// TwinCAT 3 PLC project PLC_HMI
// ProgramVersion: 3.1.4024.0
// libraries:
//   CmpBitmapPool, * (System)
//   Tc2_Standard, * (Beckhoff Automation GmbH)
//   Tc2_System, * (Beckhoff Automation GmbH)
//   Tc2_Utilities, * (Beckhoff Automation GmbH)
//   Tc3_Module, * (Beckhoff Automation GmbH)
//   VisuDialogs, * (System)
// project tree:
//   / GlobalTextList.TcGTLO, PlcTask.TcTTO, VisualizationManager.TcVMO (not stored), VISU_TASK.TcTTO
//   GVLs/ GVL.TcGVL
//   POUs/ FB_UpdateTimeStamp.TcPOU, MAIN.TcPOU, OP_BTN.TcPOU
//   VISUs/ CONFIRMATION.TcVIS, FOOTER.TcVIS, PAGE_SYSTEM.TcVIS, PAGE_RUN.TcVIS, ImagePool.TcIPO (not stored), PAGE_HOME.TcVIS, PAGE_CONTROL.TcVIS
// real-time tasks:
//   TASK PlcTask: cycle T#10ms, priority 20, ADS port 350
//   TASK VISU_TASK: cycle T#200000us, priority 30, ADS port 351

CONFIGURATION PLC_HMI
    RESOURCE PLC ON TwinCAT3
        TASK PlcTask(INTERVAL := T#10ms, PRIORITY := 20);
        TASK VISU_TASK(INTERVAL := T#200000us, PRIORITY := 30);
        PROGRAM MAIN WITH PlcTask : MAIN;
        PROGRAM VisuElems_Visu_Prg WITH VISU_TASK : VisuElems.Visu_Prg;
    END_RESOURCE
END_CONFIGURATION

// ---- GVLs/GVL.TcGVL
{attribute 'qualified_only'}
VAR_GLOBAL
	TableRecord		: ARRAY [1..5,1..7] OF STRING;
	TODAY			: WORD;
	YESTERDAY		: WORD;
	LASTMONTH		: UINT;
	LASTYEAR		: UINT;
	
	DailyCnt_FG1	: INT;
	DailyCnt_FG2	: INT;
	DailyCnt_FG3	: INT;
	DailyCnt_FG4	: INT;
	MonthCnt		: UINT;
	YearCnt			: UINT;
END_VAR

// ---- POUs/MAIN.TcPOU
PROGRAM MAIN
VAR
	fb_TimeStamp : FB_UpdateTimeStamp ();
END_VAR

// Open PLC HMI view here C:\TwinCAT\3.1\Components\Plc\Tc3PlcHmi
// Open PLC HMI web view with this link   http://127.0.0.1/Tc3PlcHmiWeb/Port_851/Visu/webvisu.htm


fb_TimeStamp();
OP_BTN();

END_PROGRAM

// ---- POUs/FB_UpdateTimeStamp.TcPOU
FUNCTION_BLOCK FB_UpdateTimeStamp
VAR_INPUT
END_VAR
VAR_OUTPUT
	FullSystemTime	: STRING;
	SystemYear		: STRING;
	SystemDate		: STRING;
	SystemTime		: STRING;
	SystemHour		: STRING;
	timeValid		: BOOL;
	day 	: ARRAY [1..7] OF BOOL;
END_VAR
VAR
	fb_LocalTime	 : FB_LocalSystemTime;
END_VAR

//  --------------------------------------------------------------- Initialize
	fb_LocalTime(
			sNetID:= , 
			bEnable:= TRUE , 
			dwCycle:= 1, 
			dwOpt:= , 
			tTimeout:= ,
			bValid=> timeValid, 
			systemTime=> , 
			tzID=> );
			
//  --------------------------------------------------------------- Set system time	
	IF fb_localTime.bValid THEN
		FullSystemTime 	:= SYSTEMTIME_TO_STRING(fb_LocalTime.systemTime);
		
		SystemYear		:= WORD_TO_STRING(fb_LocalTime.systemTime.wYear);
		SystemDate		:= WORD_TO_STRING(fb_LocalTime.systemTime.wYear);
		SystemDate		:= CONCAT(SystemDate, '.');
		SystemDate		:= CONCAT(SystemDate, WORD_TO_STRING(fb_LocalTime.systemTime.wMonth));
		SystemDate		:= CONCAT(SystemDate, '.');
		SystemDate		:= CONCAT(SystemDate, WORD_TO_STRING(fb_LocalTime.systemTime.wDay));
		
		SystemTime		:= WORD_TO_STRING(fb_LocalTime.systemTime.wHour);
		SystemTime		:= CONCAT(SystemTime, ':');
		SystemTime		:= CONCAT(SystemTime, WORD_TO_STRING(fb_LocalTime.systemTime.wMinute));
		SystemTime		:= CONCAT(SystemTime, ':');
		SystemTime		:= CONCAT(SystemTime, WORD_TO_STRING(fb_LocalTime.systemTime.wSecond));
		
		SystemHour		:= WORD_TO_STRING(fb_LocalTime.systemTime.wHour);
		
	END_IF

END_FUNCTION_BLOCK

// ---- POUs/OP_BTN.TcPOU
PROGRAM OP_BTN
VAR
	Start_btn	: BOOL;
	Start_lamp	: BOOL;
	Reset_btn	: BOOL;
	Reset_lamp	: BOOL;
	Estop_btn	: BOOL;
	Estop_lamp	: BOOL;
END_VAR

// Lamp Operation 

Start_lamp := Start_btn AND NOT Reset_btn AND NOT Estop_btn;

Estop_lamp := Estop_btn AND NOT Reset_btn;


// Lamp Reset
IF Reset_btn THEN
	Start_btn := Estop_btn := FALSE;
	Reset_lamp := TRUE;
END_IF

IF Estop_btn THEN
	Start_btn := Reset_btn := FALSE;
	Reset_lamp := FALSE;
END_IF

END_PROGRAM

// ---- GlobalTextList.TcGTLO
TEXTLIST GlobalTextList
  82 = '%s'
  902 = 'Admin'
  132 = 'ADMIN'
  997 = 'Are you Sure ?'
  180 = 'Calibration'
  3105 = 'Connect   Laser'
  1339 = 'Connect Scanner'
  395 = 'Control'
  313 = 'CONTROL PAGE'
  934 = 'Emergency Stop'
  133 = 'Home'
  266 = 'HOME PAGE'
  186 = 'Login'
  47 = 'LOGIN'
  735 = 'Logout'
  992 = 'LOGOUT'
  2441 = 'Mute\nBuzzer'
  532 = 'No'
  472 = 'None'
  30 = 'Operator'
  391 = 'OPERATOR'
  92 = 'Reset Button'
  885 = 'Run'
  192 = 'RUN PAGE'
  899 = 'Selected model'
  941 = 'Start Button'
  88 = 'System'
  451 = 'SYSTEM PAGE'
  608 = 'WARNING'
  412 = 'Yes'
END_TEXTLIST

// ---- VISUs/CONFIRMATION.TcVIS
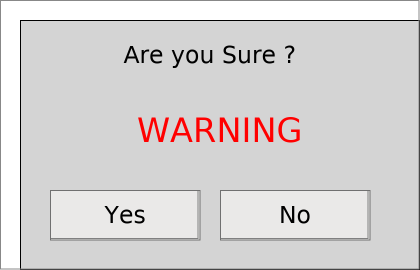
VISUALIZATION CONFIRMATION  // 420x270
VAR_IN_OUT
	result : STRING;
END_VAR
    Rectangle (20,20 400x250)
    Button (50,190 150x50), "Yes"
        toggle OP_BTN.Start_btn
        OnMouseClick: CloseDialog Dialog=CONFIRMATION, Result=Yes, NumpadKeypadSet=True
    Label (85,30 250x50), "Are you Sure ?"
    Button (220,190 150x50), "No"
        OnMouseClick: CloseDialog Dialog=CONFIRMATION, Result=No, NumpadKeypadSet=True
    Textfield (20,100 400x60), "WARNING"
END_VISUALIZATION

// ---- VISUs/FOOTER.TcVIS
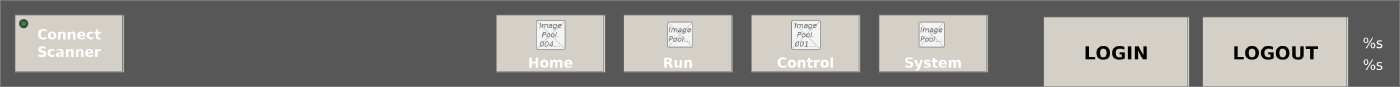
VISUALIZATION FOOTER  // 1920x120
    Textfield (1700,70 200x40), "%s", text variable: MAIN.fb_TimeStamp.SystemDate
    Textfield (1700,40 200x40), "%s", text variable: MAIN.fb_TimeStamp.SystemTime
    Group (855,20 150x80)
        OnMouseClick: change screen: PAGE_RUN
        Button (0,0 150x80), "Run"
        Image (60,10 35x35), image: ImagePool.003-play-button-arrowhead
    Group (1030,20 150x80)
        OnMouseClick: change screen: PAGE_CONTROL
        Button (0,0 150x80), "Control"
        Image (55,8 40x40), image: ImagePool.001-gear
    Group (680,20 150x80)
        OnMouseClick: change screen: PAGE_HOME
        Button (0,0 150x80), "Home"
        Image (55,8 40x40), image: ImagePool.004-home
    Group (1205,20 150x80)
        OnMouseClick: change screen: PAGE_SYSTEM
        Button (0,0 150x80), "System"
        Image (55,10 35x35), image: ImagePool.002-folder
    Button (20,20 150x80), "Connect Scanner"
    Lamp1 (25,25 15x15), style: Lamp-Lamp1-Green
    Group (1431,23 293x60)
        Button (218,0 200x100), "LOGOUT"
            OnMouseClick: VisuUserMgmt Type=Logout
        Button (0,0 200x100), "LOGIN"
            OnMouseClick: VisuUserMgmt Type=Login
END_VISUALIZATION

// ---- VISUs/PAGE_SYSTEM.TcVIS
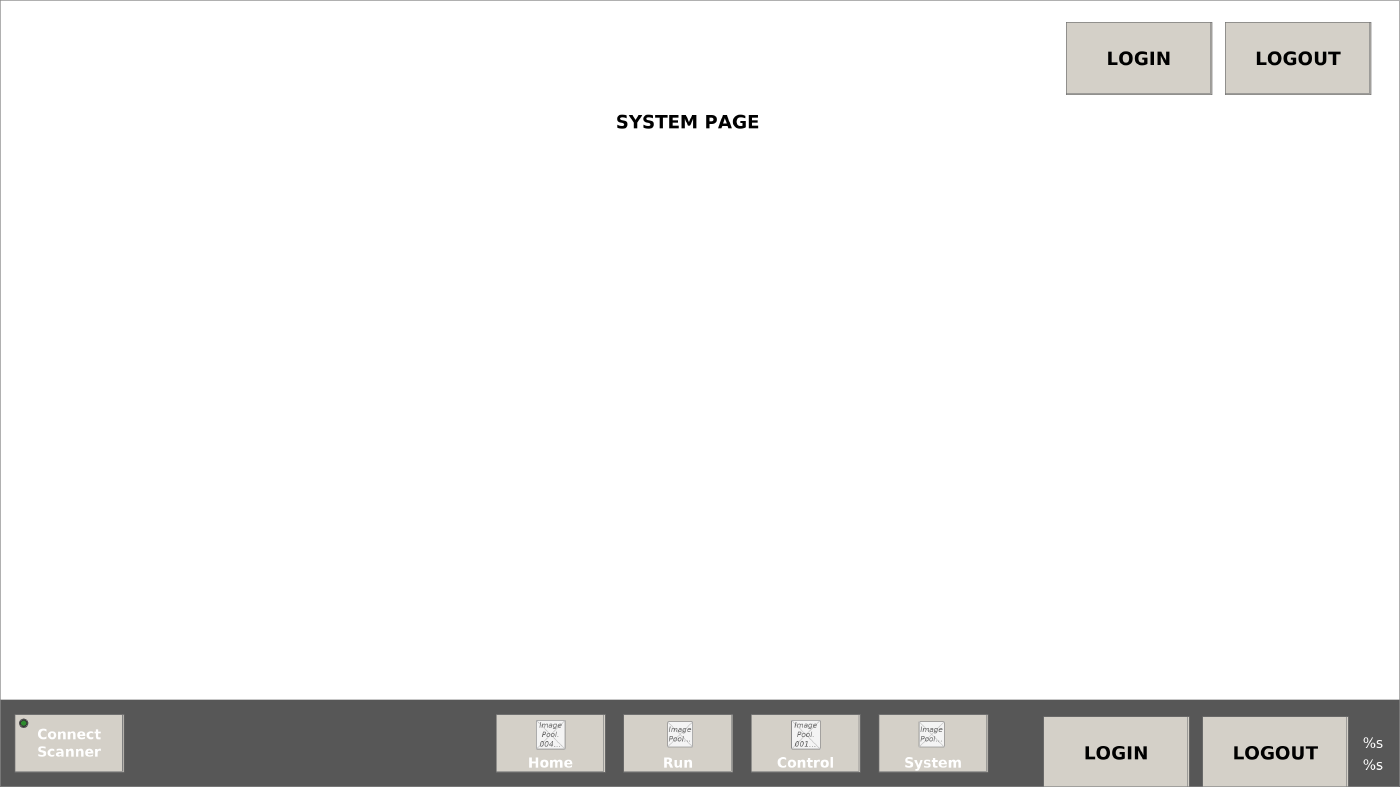
VISUALIZATION PAGE_SYSTEM  // 1920x1080, background image ImagePool.Grey_Gradient
    Button (1462,30 200x100), "LOGIN"
        OnMouseClick: VisuUserMgmt Type=Login
    Button (1680,30 200x100), "LOGOUT"
        OnMouseClick: VisuUserMgmt Type=Logout
    Frame (0,960 1920x120)
        shows FOOTER()
    Label (708,109 470x116), "SYSTEM PAGE"
END_VISUALIZATION

// ---- VISUs/PAGE_RUN.TcVIS
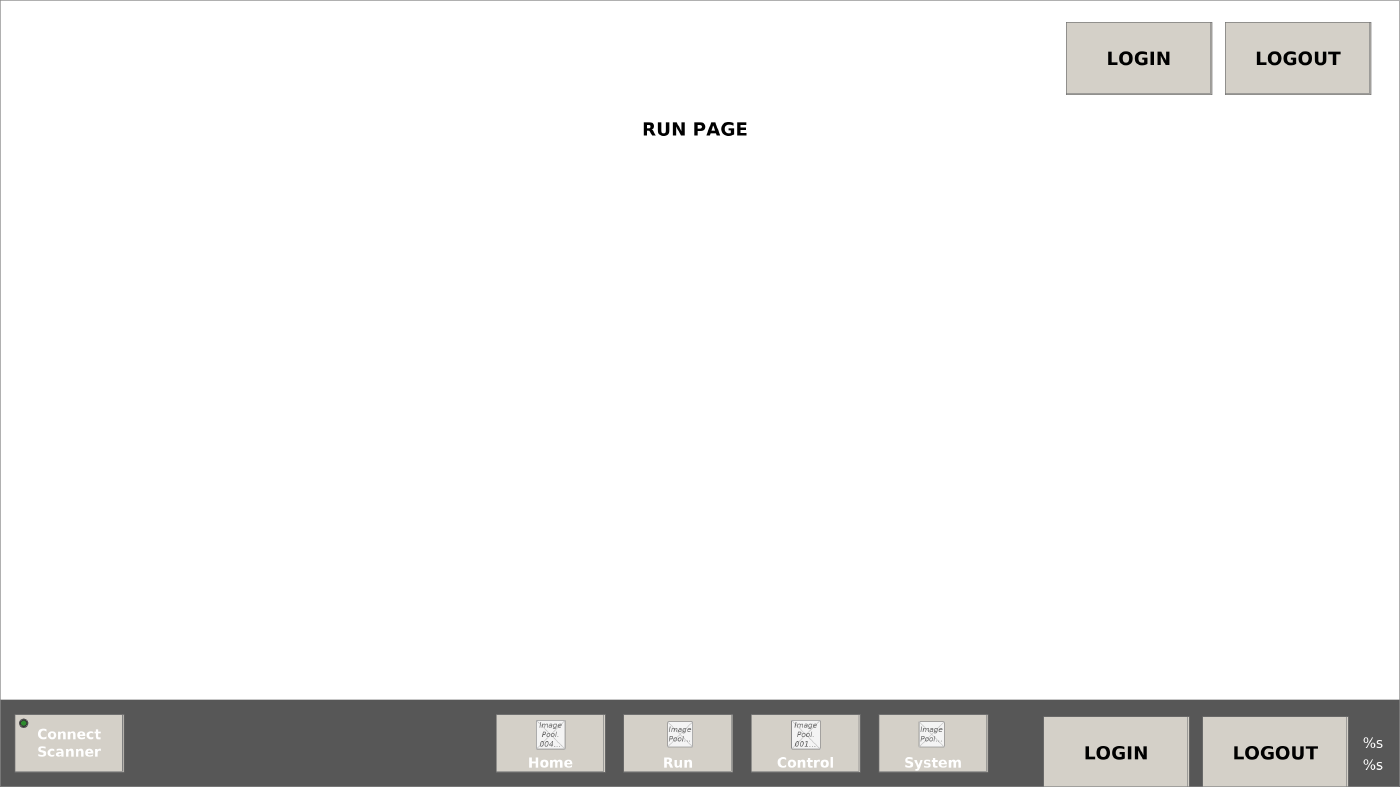
VISUALIZATION PAGE_RUN  // 1920x1080, background image ImagePool.Grey_Gradient
    Button (1462,30 200x100), "LOGIN"
        OnMouseClick: VisuUserMgmt Type=Login
    Button (1680,30 200x100), "LOGOUT"
        OnMouseClick: VisuUserMgmt Type=Logout
    Frame (0,960 1920x120)
        shows FOOTER()
    Label (718,119 470x116), "RUN PAGE"
END_VISUALIZATION

// ---- VISUs/PAGE_HOME.TcVIS
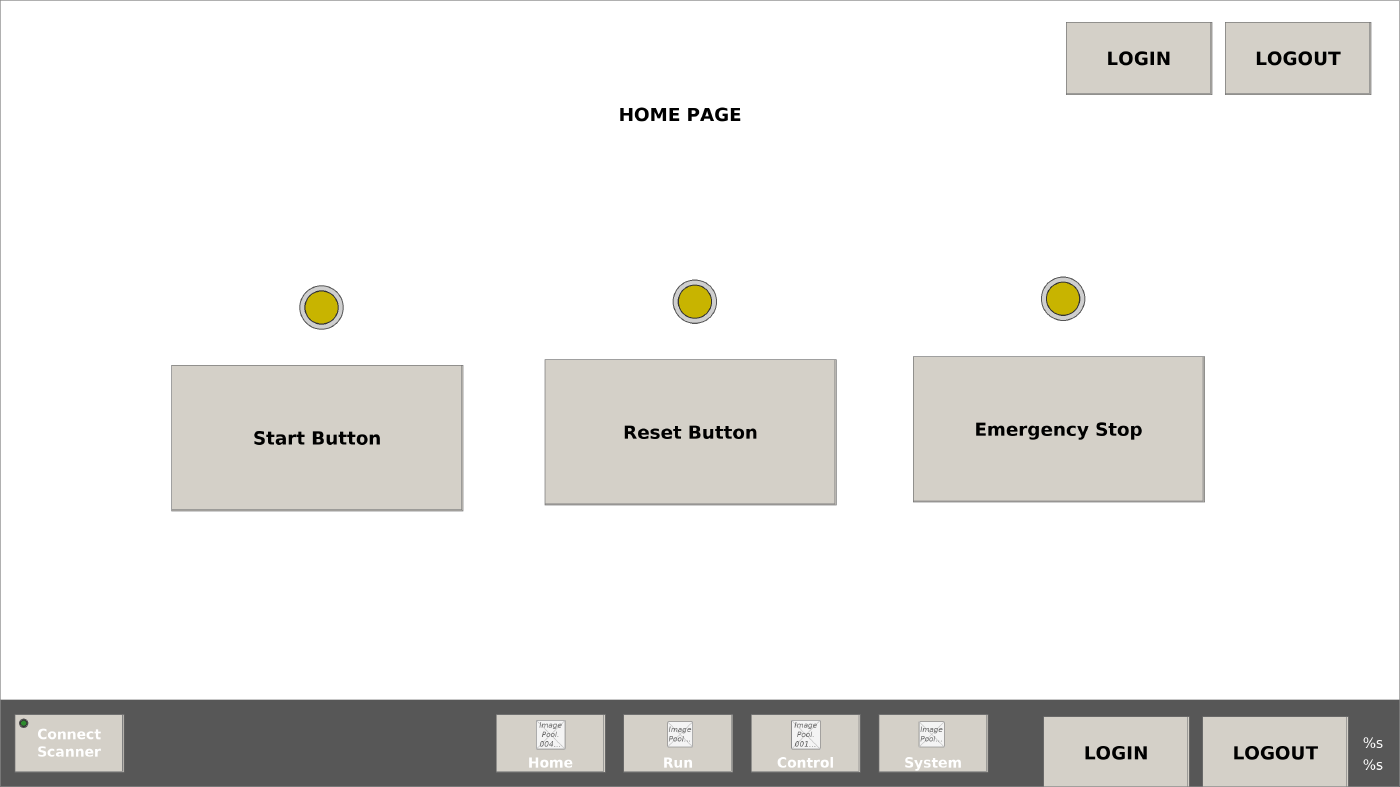
VISUALIZATION PAGE_HOME  // 1920x1080, background image ImagePool.Grey_Gradient
    Button (235,501 400x200), "Start Button"
        OnMouseClick: OpenDialog Dialog=CONFIRMATION, OpenModal=True, OpenCentered=True
    Lamp1 (406,387 70x70), variable: OP_BTN.Start_lamp, style: Lamp-Lamp1-Yellow
    Button (747,493 400x200), "Reset Button"
        tap OP_BTN.Reset_btn
    Lamp1 (918,379 70x70), variable: OP_BTN.Reset_lamp, style: Lamp-Lamp1-Yellow
    Button (1252,489 400x200), "Emergency Stop"
        toggle OP_BTN.Estop_btn
    Lamp1 (1423,375 70x70), variable: OP_BTN.Estop_lamp, style: Lamp-Lamp1-Yellow
    Button (1462,30 200x100), "LOGIN"
        OnMouseClick: VisuUserMgmt Type=Login
    Button (1680,30 200x100), "LOGOUT"
        OnMouseClick: VisuUserMgmt Type=Logout
    Frame (0,960 1920x120)
        shows FOOTER()
    Label (698,99 470x116), "HOME PAGE"
END_VISUALIZATION

// ---- VISUs/PAGE_CONTROL.TcVIS
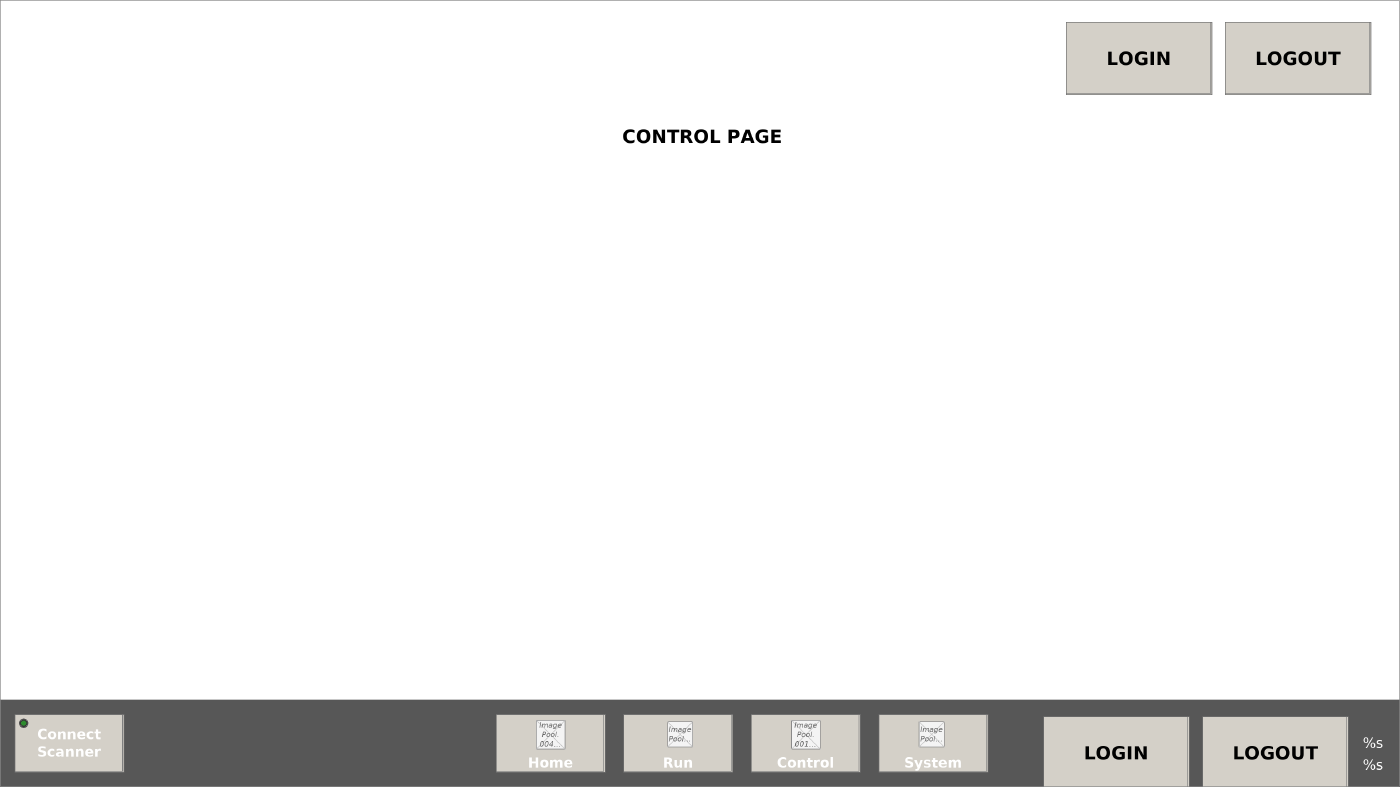
VISUALIZATION PAGE_CONTROL  // 1920x1080, background image ImagePool.Grey_Gradient
    Button (1462,30 200x100), "LOGIN"
        OnMouseClick: VisuUserMgmt Type=Login
    Button (1680,30 200x100), "LOGOUT"
        OnMouseClick: VisuUserMgmt Type=Logout
    Frame (0,960 1920x120)
        shows FOOTER()
    Label (728,129 470x116), "CONTROL PAGE"
END_VISUALIZATION
